// TIA Portal V19 export
TYPE "LEXCHANGETRAY_typeHandlingXyz_signalTM_Monitor"
// stored: Access Published
   STRUCT
      simulationed : Bool;
      GripperCylinderHomePositionDetectionU2EM4_1 : Bool;
      gripperCylinderWorkPositionDetectionOfSmallCellU2EM4_2 : Bool;
      withOrWithoutCellDetectionU2EM4_2 : Bool;
      GripperCylinderHomePositionDetectionU2EM4_3 : Bool;
      yaxlEmotorOrgU2EM4 : Bool;
      yaxlEmotorPotU2EM4 : Bool;
      gripperCylinderWorkPositionDetectionOfSmallCellU2EM4_4 : Bool;
      handlingCollisionAvoidance2U2EM4 : Bool;
      gripperCylinderWorkPositionDetectionOfSmallCellU2EM4_3 : Bool;
      gripperCylinderWorkPositionDetectionOfBigCellU2EM4_3 : Bool;
      gripperCylinderWorkPositionDetectionOfBigCellU2EM4_2 : Bool;
      gripperCylinderWorkPositionDetectionOfBigCellU2EM4_1 : Bool;
      xaxlEmotorPotU2EM4 : Bool;
      zaxlEmotorNotU2EM4 : Bool;
      cellFoolproof4U2EM4 : Bool;
      withOrWithoutCellDetectionU2EM4_3 : Bool;
      cellFoolproof1U2EM4 : Bool;
      xaxlEmotorOrgU2EM4 : Bool;
      GripperCylinderHomePositionDetectionU2EM4_2 : Bool;
      xaxlEmotorNotU2EM4 : Bool;
      handlingCollisionAvoidance4U2EM4 : Bool;
      handlingCollisionAvoidance3U2EM4 : Bool;
      zaxlEmotorPotU2EM4 : Bool;
      cellFoolproof3U2EM4 : Bool;
      zaxlEmotorOrgU2EM4 : Bool;
      yaxlEmotorNotU2EM4 : Bool;
      handlingCollisionAvoidance1U2EM4 : Bool;
      cellFoolproof2U2EM4 : Bool;
      gripperCylinderWorkPositionDetectionOfSmallCellU2EM4_1 : Bool;
      withOrWithoutCellDetectionU2EM4_4 : Bool;
      gripperCylinderWorkPositionDetectionOfBigCellU2EM4_4 : Bool;
      GripperCylinderHomePositionDetectionU2EM4_4 : Bool;
      withOrWithoutCellDetectionU2EM4_1 : Bool;
   END_STRUCT;
END_TYPE
